// TwinCAT 3 PLC project EnOcean_Sample_CX9020_1
// libraries:
//   Tc2_EnOcean, * (Beckhoff Automation GmbH)
//   Tc2_Standard, * (Beckhoff Automation GmbH)
//   Tc2_System, * (Beckhoff Automation GmbH)
//   Tc3_Module, * (Beckhoff Automation GmbH)
// project tree:
//   Global Variables/ Globale_Variablen.TcGVL, Variablen_Konfiguration.TcGVL (not stored)
//   POUs/ MAIN.TcPOU
//   / Standard.TcTTO (not stored)

// ---- Global Variables/Globale_Variablen.TcGVL
{attribute 'Tc2GvlVarNames'}
VAR_GLOBAL
	st6581Input  AT %I* : KL6581_Input;
	st6581Output AT %Q* : KL6581_Output;
	stKL6581            : STR_KL6581;
END_VAR

// ---- POUs/MAIN.TcPOU
PROGRAM MAIN
VAR
	fbKL6581			: FB_KL6581;

	fbRec_RPS_Switch	: FB_Rec_RPS_Switch;
	dwId				: DWORD := 1059793;
	stEnOceanSwitch		: STR_EnOceanSwitch;
	bReady				: BOOL;
	bBusy				: BOOL;
	bError				: BOOL;
	iErrorId			: INT;
END_VAR

fbKL6581(bInit := TRUE, stKL6581_in := st6581Input, stKL6581_out := st6581Output); // FB_KL6581
bReady := fbKL6581.bReady;
bBusy := fbKL6581.bBusy;
bError := fbKL6581.bError;
iErrorId := fbKL6581.iErrorID;
stKL6581 := fbKL6581.str_KL6581;
fbRec_RPS_Switch(str_KL6581 := stKL6581, dw_ID := dwId); // FB_Rec_RPS_Switch
stEnOceanSwitch := fbRec_RPS_Switch.str_EnOceanSwitch;

END_PROGRAM
